(* IEC 61131-3 sources: Std_PalletMover/Class/CanDriverCPU, 1 file *)

(* ---- CanDriverCPU.st ---- *)
(*!
<Class
	Name               = "CanDriverCPU"
	Revision           = "0.2"
	RealtimeTask       = "false"
	CyclicTask         = "false"
	BackgroundTask     = "false"
	Sigmatek           = "false"
	OSInterface        = "false"
	HighPriority       = "false"
	Automatic          = "false"
	UpdateMode         = "Prescan"
	SharedCommandTable = "true"
	Objectsize         = "(540,240)">
	<Channels>
		<Server Name="CanBus" Visualized="true" Initialize="true" WriteProtected="true" Retentive="false" Comment="which CanbusSystem [1,2,...](as initvalue)"/>
		<Client Name="_CanLib0" Required="true" Internal="true"/>
		<Client Name="To_Can" Required="false" Internal="false" Comment="is connected automatically"/>
	</Channels>
	<Network Name="CanDriverCPU">
		<!-- List of Components in this network -->
		<Components>
			<Object
				Name       = "_base"
				Class      = "CanDriverBase"
				Position   = "(570,120)"
				Visualized = "true">
				<Channels>
					<Server Name="Command"/>
					<Server Name="ErrCntr"/>
					<Server Name="Status"/>
					<Client Name="CanChannel"/>
					<Client Name="cBaudrate"/>
					<Client Name="IrqChannel"/>
				</Channels>
			</Object>
			<Object
				Name       = "_CanLib0"
				Class      = "_CanLib"
				Position   = "(180,120)"
				Visualized = "true">
				<Channels>
					<Server Name="CanBus" Value="1"/>
					<Server Name="Command"/>
					<Client Name="To_Can"/>
				</Channels>
			</Object>
		</Components>
		<Comments>
		</Comments>
		<!-- List of Connections in this network -->
		<Connections>
			<Connection Source="_base.CanChannel" Destination="_CanLib0.Command" Vertices="(570,210),(510,210),"/>
			<Connection Source="_base.cBaudrate" Destination="this.cBaudrate" Vertices="(570,270),(38,210),"/>
			<Connection Source="_base.IrqChannel" Destination="this.IrqChannel" Vertices="(570,330),(38,270),"/>
			<Connection Source="this.Command" Destination="_base.Command" Vertices="(1132,210),(960,210),"/>
			<Connection Source="this.Status" Destination="_base.Status" Vertices="(1132,270),(960,270),"/>
			<Connection Source="this._CanLib0" Destination="_CanLib0.Command"/>
			<Connection Source="this.ErrCntr" Destination="_base.ErrCntr" Vertices="(1132,330),(960,330),"/>
			<Connection Source="_CanLib0.To_Can" Destination="this.To_Can" Vertices="(180,210),(38,390),"/>
			<Connection Source="this.CanBus" Destination="_CanLib0.CanBus" Vertices="(1132,390),(510,270),"/>
		</Connections>
		<!-- Headerfiles -->
		<Options>
		</Options>
	</Network>
</Class>
*)
#pragma using CanDriverBase

CanDriverCPU : CLASS
: CanDriverBase
  //Servers:
	CanBus 	: SvrCh_DINT;
  //Clients:
	_CanLib0 	: CltChCmd__CanLib;
	To_Can 	: CltChCmd__Can;
  //Variables:
  //Functions:

	FUNCTION VIRTUAL GLOBAL CanBus::Read
		VAR_OUTPUT
			output (EAX) 	: DINT;
		END_VAR;
  //Tables:
	FUNCTION @STD
		VAR_OUTPUT
			ret_code	: CONFSTATES;
		END_VAR;
	FUNCTION GLOBAL TAB @CT_;
END_CLASS;

#pragma using _CanLib
#pragma usingLtd _Can

FUNCTION VIRTUAL GLOBAL CanDriverCPU::CanBus::Read
	VAR_OUTPUT
		output (EAX) 	: DINT;
	END_VAR

	CanBus := _CanLib0.CanBus.Read();
	output := CanBus;

END_FUNCTION
